FUNCTION_BLOCK FB_InfoConnection
VAR_INPUT
	stInfoData	:ST_InfoDataConnection;
END_VAR
VAR_OUTPUT
	sState		:STRING;
	sDiag		:STRING;
	bChannel1	:BOOL;
	bChannel2	:BOOL;
	bChannel3	:BOOL;
	bChannel4	:BOOL;
END_VAR

IF stInfoData.usiMapState = 100 THEN
	sState:='State Reset';
ELSIF stInfoData.usiMapState = 101 THEN
	sState:='State Session';
ELSIF stInfoData.usiMapState = 102 THEN
	sState:='State Connection';
ELSIF stInfoData.usiMapState = 103 THEN
	sState:='State Parameter';
ELSIF stInfoData.usiMapState = 104 THEN
	sState:='State Data';
ELSIF stInfoData.usiMapState = 105 THEN
	sState:='State Shutdown';
ELSE
	sState:='Error';
END_IF

IF stInfoData.usiMapDiag = 0 THEN
	sDiag:='No error';
ELSIF	stInfoData.usiMapDiag.0 = TRUE THEN
	sDiag:='Invalid Command';
ELSIF	stInfoData.usiMapDiag.1 = TRUE THEN
	sDiag:='Unknown Command';
ELSIF	(stInfoData.usiMapDiag.1 AND stInfoData.usiMapDiag.0)= TRUE THEN
	sDiag:='Invalid Connection ID';
ELSIF	 stInfoData.usiMapDiag.2= TRUE THEN
	sDiag:='Invalid CRC';
ELSIF	(stInfoData.usiMapDiag.0 AND stInfoData.usiMapDiag.2)= TRUE THEN
	sDiag:='Watchdog expired';
ELSIF	(stInfoData.usiMapDiag.1 AND stInfoData.usiMapDiag.2)= TRUE THEN
	sDiag:='Invalid FSoE address';
ELSIF	(stInfoData.usiMapDiag.0 AND stInfoData.usiMapDiag.1 AND stInfoData.usiMapDiag.2)= TRUE THEN
	sDiag:='Invalid data';
ELSIF	stInfoData.usiMapDiag.3= TRUE THEN
	sDiag:='Invalid Com.-Parameter length';
ELSIF	(stInfoData.usiMapDiag.0 AND stInfoData.usiMapDiag.3)= TRUE THEN
	sDiag:='Invalid Com.-Parameter ';
ELSIF	(stInfoData.usiMapDiag.1 AND stInfoData.usiMapDiag.3)= TRUE THEN
	sDiag:='Invalid User.-Parameter length';
ELSIF	(stInfoData.usiMapDiag.0 AND stInfoData.usiMapDiag.1 AND stInfoData.usiMapDiag.3)= TRUE THEN
	sDiag:='Invalid User.-Parameter ';
ELSIF	(stInfoData.usiMapDiag.2 AND stInfoData.usiMapDiag.3)= TRUE THEN
	sDiag:='FSoE Master Reset  ';
ELSIF	stInfoData.usiMapDiag.4= TRUE THEN
	sDiag:='Error by FSoE Slave detected';
ELSIF	stInfoData.usiMapDiag.5= TRUE THEN
	sDiag:='FSoE Slave reports Failsafe value active';
ELSIF	stInfoData.usiMapDiag.6= TRUE THEN
	sDiag:='StartUp';
ELSIF	stInfoData.usiMapDiag.7= TRUE THEN
	sDiag:='FSoE Master reports Failsafe value active';
ELSE
	sDiag:='Error';
END_IF

(*Signals*)
bChannel1 := stInfoData.bySignal.0;
bChannel2 := stInfoData.bySignal.1;
bChannel3 := stInfoData.bySignal.2;
bChannel4 := stInfoData.bySignal.3;

END_FUNCTION_BLOCK

(* stored: Version 1.1.0.1, ProductVersion 3.1.4024.12
   POU FB_InfoConnection: Id {20866d00-a67f-4183-9603-a0bbdd91ae1d}, SpecialFunc None *)
